(* PLC project rien2, Dassault Systèmes ControlBuild 2024x Refresh1 *)
(* stored: creationDateTime 2024-03-14T09:59:36-01:00 *)

FUNCTION_BLOCK st1


ACTION C_source_code:

END_ACTION
END_FUNCTION_BLOCK

PROGRAM aaa1

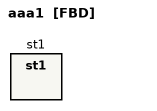
(* FBD diagram, written out as Structured Text *)
st1();
END_PROGRAM

PROGRAM my_app.rien2

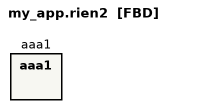
(* FBD diagram, written out as Structured Text *)
aaa1();
END_PROGRAM
